Staubli VAL3: putEx2.pgx

public program putEx2(string sX, num nY, string sText)
  local num nX
begin
  // Displays a text at [left/center/right] horizontal position
  //
  // The cursor is positioned on the character after the last character of
  // the message displayed
  //
  // copyright (c) 2020 victortorreslopez
  //
  // GNU General Public License
  //
  // Parameters
  // - sX: horizontal alignment (left, center, right)
  // - nY: cursor row (0 to 13)
  // - sText: character string type expression
  //
  // Locals variables
  // - nX: cursor column (0 to 39)
  //
  // Version history
  // ---------------
  // 0.0, 2020/11/21, VTL: alfa release from "_put"

  call lower(sX)

  if len(sText) > 40
    nX = 0
  else
    if sX == "right"
      nX = 40 - len(sText)
    elseIf sX == "center"
      nX = (40 - len(sText)) / 2
    elseIf sX == "left"
      nX = 0
    endIf
  endIf

  gotoxy(nX, nY)
  put(sText)
end
